PROGRAM MAIN
VAR
    fbPersistentDataStorage : FB_PersistentDataStorage;
	{attribute 'pytmc' := '
		axis-link: GVL_Axes.Axes[1]
		pv: TST:MOTION:SLITX
	'}
   	slitX : FB_MotionStageNC(	sName := 'slitX',
                                        AxisRef := GVL_Axes.Axes[1],
                                        iPersistentDataStorage := fbPersistentDataStorage
                                    ) ;
	{attribute 'pytmc' := '
		axis-link: GVL_Axes.Axes[2]
		pv: TST:MOTION:SLITY
	'}
   	slitY : FB_MotionStageNC(	sName := 'slitY',
                                        AxisRef := GVL_Axes.Axes[2],
                                        iPersistentDataStorage := fbPersistentDataStorage
                                    ) := (EnableMode:=E_StageEnableMode.ALWAYS);
	{attribute 'pytmc' := '
		axis-link: GVL_Axes.Axes[3]
		pv: TST:MOTION:SLITZ
	'}
   	slitZ : FB_MotionStageNC(	sName := 'slitZ',
                                        AxisRef := GVL_Axes.Axes[3],
                                        iPersistentDataStorage := fbPersistentDataStorage
                                    ) ;
   	dummy : FB_MotionStageNC(	sName := 'dummy',
                                        AxisRef := GVL_Axes.Axes[4],
                                        iPersistentDataStorage := fbPersistentDataStorage
                                    ) ;
END_VAR

fbPersistentDataStorage();
slitX();
slitY();
slitZ();
dummy();

END_PROGRAM

(* stored: Version 1.1.0.1
   POU MAIN: Id {7ddf7142-3738-4120-8059-c5d2220b5135}, SpecialFunc None *)
